{attribute 'Tc2GvlVarNames'}
{attribute 'strict'}
//Tipologia Di Presa dell' Elemento da parte dell'End Effector
TYPE e_Tipo_ChiusuraAsseK :
(
	KNOTDEFINEDMODE	:= -1,//Prelievo con ventose
	KSUCTIONMODE	:= 0,//Prelievo con ventose
	KPOSITIONMODE	:= 1,//Prelievo a quota
	KTORQUEMODE		:= 2//Prelievo con coppia
);
END_TYPE
//  KNOTDEFINEDMODE = '-1'

(* stored: Version 1.1.0.1, ProductVersion 3.1.4024.11
   EnumerationTextList e_Tipo_ChiusuraAsseK: Id {57d10f3b-1ef8-4de4-8a15-7c7e78fa4727} *)
